Staubli VAL3: stop.pgx

public program stop()
  local num l_nI
begin
  //-----------------------------------------------------------------------
  //Header begin
  //Description of program
  //  Release all IDs.
  //  This routine should be called once when ending main application.
  //
  //History
  //  Creation : 12-12 - CROC
  //Header end
  //-----------------------------------------------------------------------
  //Reset all cameras in the array
  for l_nI=0 to size(cCamera)-1
    cCamera[l_nI].bConnected=false
  endFor
  resetMotion()
  disablePower()
  vbleu=false
  vvert=false
  vorange=false
  vrouge=false
  nbPoint=0
end
